PROGRAM SizeCheck
VAR
	bundleSize : ULINT;
	adsDataSize : ULINT;
	tcpDataSize : ULINT;
	
	thousandByteSize : ULINT;
	buffer : ARRAY[0..1000] OF BYTE;
	
	bitArr : ARRAY[1..64] OF ONE_BIT;
	bitArrSize : ULINT;
END_VAR

bundleSize := SIZEOF(Bundle);
adsDataSize := SIZEOF(AdsData);
tcpDataSize := SIZEOF(TcpData);

thousandByteSize := SIZEOF(buffer);

bitArrSize := SIZEOF(bitArr);

END_PROGRAM

(* stored: Version 1.1.0.1, ProductVersion 3.1.4024.11
   POU SizeCheck: Id {58756afd-ee77-4842-8005-9b6b1a222eca}, SpecialFunc None *)
